(* PLC project  *)

CONFIGURATION EL1809
END_CONFIGURATION
